{attribute addProperty BoxType "EM7004-0000-9995"}
{attribute addProperty Id "CtrlAT %Q*UINT1621ValueAT %Q*UINT1622"}
{attribute addProperty CRC "110769869"}
{attribute addProperty SizeInBites "32"}
{attribute addProperty SizeInBytes "4"}
TYPE Encoder_Channel_069A36CD :
STRUCT
	{attribute addProperty Name "Ctrl"}
	Ctrl AT %Q* : UINT;
	{attribute addProperty Name "Value"}
	Value AT %Q* : UINT;
END_STRUCT
END_TYPE

(* stored: Version 1.2.0.0, ProductVersion 3.1.4024.9
   DUT Encoder_Channel_069A36CD: Id {ff231a51-e07f-4e0d-8c3f-5849500c1d3a} *)
